Fanuc KAREL source: kt00483.KL

-- PROVISIONAL review KL for V940-1; original PC SHA256 52682d885713f2f0d50bd8a33cbb0cfd443cd6f42a4543a5a36c2b83162f3db5
-- Incomplete behavior may be omitted. Consult companion uncertainty JSON. Do not deploy.
PROGRAM KT00483
%NOLOCKGROUP
VAR
  OUT : BOOLEAN
-- UNRESOLVED_DECL P1 type=000101
-- UNRESOLVED_DECL P2 type=000106
BEGIN
  -- V9_ZERO_TABLE_METADATA_HINT layout=0001; no indexed target words; source/name/runtime held
  -- UNRESOLVED_PC offsets 5-20; opcodes 2E,22,32,35
  -- UNRESOLVED_PC offsets 25-53; opcodes 49,49,7E,AC,23
  -- UNRESOLVED_PC offsets 58-62; opcodes 7F
END KT00483
